TYPE PVType :
(
	PVType_Default := 0, // 常规的PV阀
	PVType_VAT := 1, // VAT
	PVType_Other := 2 // Other
)UINT;
END_TYPE

(* stored: Version 1.1.0.1, ProductVersion 3.1.4024.4
   DUT PVType: Id {50e678ca-4b25-4817-abdd-e7774a1eda0b} *)
